Staubli VAL3: D_ABZ_01.pjx

Parameters version=s7.6 stackSize=5000 millimeterUnit=true
Program file=_DetectIOEdge.pgx
Program file=create.pgx
Program file=encoder.pgx
Program file=getResolution.pgx
Program file=getStatus.pgx
Program file=getValue.pgx
Program file=init.pgx
Program file=isLatched.pgx
Program file=kill.pgx
Program file=reset.pgx
Program file=resetLatch.pgx
Program file=setResolution.pgx
Program file=start.pgx
Program file=stop.pgx
Data file=D_ABZ_01.dtx
